///Automatically generated by BoxConfigurator 
VAR_GLOBAL
	fbSG_001_Emulation                : FB_ProBOXSG_Emulation;
	fbSG_002_Emulation                : FB_ProBOXSG_Emulation;
END_VAR

(* stored: Version 1.1.0.1, ProductVersion 3.1.4024.9
   GVL GroupsEmulation: Id {6ca26e40-d19e-43b0-af11-c40cc36f511d} *)
